(*
	RJM Maszyny sp. z o.o.
	autor 	: Rafał Osajda
	data	: 02.02.2024
	TC		: 3.1 4024.54
	wersja	: 0.0.1.0	: pełna obsługa

	Obsługa elektrozaworu do sterowania siłownikiem pneumatycznym.sterowanie 5 na 2 2 cewki
*)
FUNCTION_BLOCK FB_Elektrozawor_5na2_2Cewki EXTENDS FB_Electrovalve

METHOD FB_init : BOOL
VAR_INPUT
	bInitRetains : BOOL; // if TRUE, the retain variables are initialized (warm start / cold start)
	bInCopyCode : BOOL;  // if TRUE, the instance afterwards gets moved into the copy code (online change)
END_VAR
THIS^.eRodzaj			:= E_ElectrovalveType.C2_5na2;
END_METHOD

(*
	RJM Maszyny sp. z o.o.
	autor 	: Rafał Osajda
	data	: 21.02.2024
	TC		: 3.1 4024.54
	wersja	: 0.0.1.0	: pełna obsługa

	Ustawienie odpowiednich wyjść
*)
METHOD Steruj : BOOL
VAR_INPUT
	eAkcja									: E_ElectrovalveAction;
END_VAR
CASE eAkcja OF
	E_ElectrovalveAction.e_EL_Wyj4_Wylacz	:
		bCewkaA								:= FALSE;
	E_ElectrovalveAction.e_EL_Wyj4_Wlacz	:
		bCewkaA								:= TRUE;
		bCewkaB								:= FALSE;
	E_ElectrovalveAction.e_EL_Wyj2_Wylacz	:
		bCewkaB								:= FALSE;
	E_ElectrovalveAction.e_EL_Wyj2_Wlacz	:
		bCewkaB								:= TRUE;
		bCewkaA								:= FALSE;
	E_ElectrovalveAction.e_EL_DoPoczatku	:
		bCewkaA								:= FALSE;
		bCewkaB								:= TRUE;
	E_ElectrovalveAction.e_EL_DoKonca		:
		bCewkaA								:= TRUE;
		bCewkaB								:= FALSE;
	E_ElectrovalveAction.e_EL_Reset			:
		bCewkaA								:= FALSE;
		bCewkaB								:= FALSE;
	E_ElectrovalveAction.e_El_Wlacz			:
		bCewkaA								:= TRUE;
		bCewkaB								:= TRUE;
	E_ElectrovalveAction.e_El_Wylacz		:
		bCewkaA								:= FALSE;
		bCewkaB								:= FALSE;	
END_CASE
END_METHOD

END_FUNCTION_BLOCK

(* stored: Version 1.1.0.1
   POU FB_Elektrozawor_5na2_2Cewki: Id {d6f8f273-ad99-08b4-23eb-da22e027bbb8}, SpecialFunc None
   Method FB_init: Id {ce8e6432-4518-46d2-b1f1-ff2916732c90}
   Method Steruj: Id {6d759c47-679a-0364-19c6-561e5615d5fc} *)
